(* CODESYS project CodesysTesting

Project tree, tasks and I/O mapping:
  Device : CODESYS Control Win V3 x64, 3S - Smart Software Solutions GmbH, version 3.5.19.50
    application Application
      libraries: Standard, 3.5.18.0 (System)
      task MainTask (cyclic, interval t#20ms, priority 1) calls PLC_PRG
      task VISU_TASK (cyclic, interval 100 ms, priority 31) calls VisuElems.Visu_Prg
      program PLC_PRG [ST]
      visualisation Visualization
  text list GlobalTextList
*)

// Device/Application/PLC_PRG
PROGRAM PLC_PRG
VAR
	i: INT;
END_VAR

i := i + 1;

END_PROGRAM

// Device/Application/Visualization
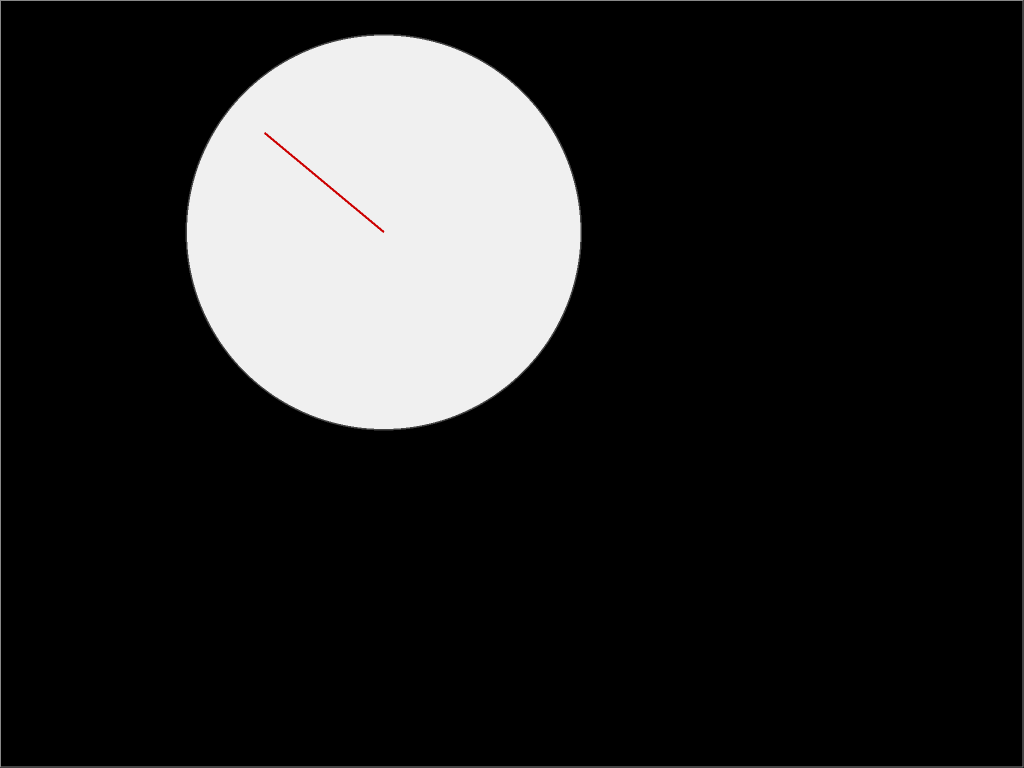
VISUALIZATION Visualization  // 1024x768
    Meter360 (157,34 453x396), value: PLC_PRG.i, style: Meter-Meter360-Gray, scale format: %.1f, scale 0..1000
END_VISUALIZATION
